% RSLogix 500 project Project_8.RSS, saved by version 8.30.00.16 %
PROJECT "UNTITLED"    % processor: Bul.1763 MicroLogix 1100 Series B %

PROGRAM FILES
  LAD 2 "MAIN"  4 rungs
  LAD 3 "IO"  3 rungs
  LAD 4 "CTL4%-15%"  7 rungs
  LAD 5 "CTL15%-30%"  7 rungs

DATA FILES
  O0 OUTPUT  4 elements
  I1 INPUT  6 elements
  S2 STATUS  66 elements
  B3 BINARY  3 elements
  T4 TIMER  4 elements
  C5 COUNTER  1 elements
  R6 CONTROL  1 elements
  N7 INTEGER  7 elements
  F8 FLOAT  1 elements

LADDER 2 "MAIN"
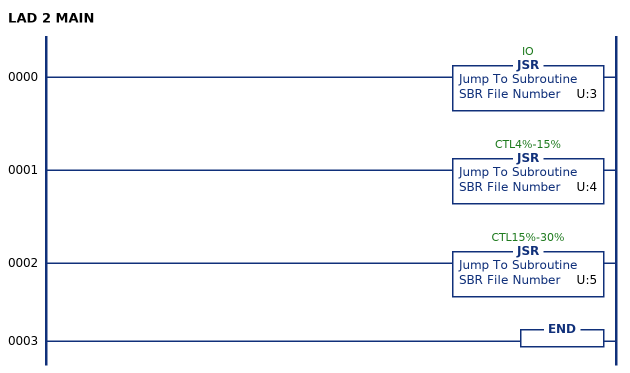
% Rung: 0 %
SOR JSR U:3 EOR
%   U:3  "IO" %
% Rung: 1 %
SOR JSR U:4 EOR
%   U:4  "CTL4%-15%" %
% Rung: 2 %
SOR JSR U:5 EOR
%   U:5  "CTL15%-30%" %
% Rung: 3 %
SOR END EOR

LADDER 3 "IO"
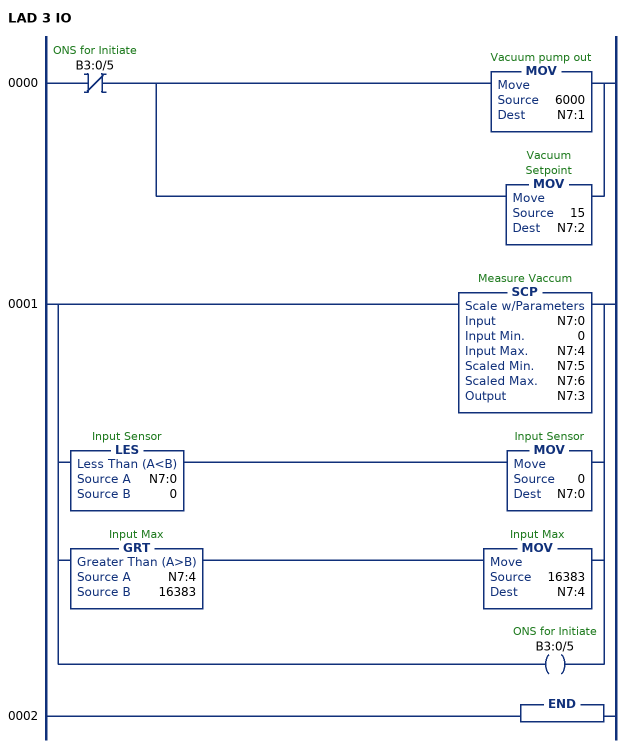
% Rung: 0 %
SOR XIO B3:0/5 BST MOV 6000 N7:1 NXB MOV 15 N7:2 BND EOR
%   B3:0/5  "ONS for Initiate" %
%   N7:1  "Vacuum pump out" %
%   N7:2  "Vacuum Setpoint" %
% Rung: 1 %
SOR BST SCP N7:0 0 N7:4 N7:5 N7:6 N7:3 NXB LES N7:0 0 MOV 0 N7:0 NXB GRT N7:4 16383 MOV 16383 N7:4 NXB OTE B3:0/5 BND EOR
%   N7:0  "Input Sensor" %
%   N7:4  "Input Max" %
%   N7:5  "Scale Min" %
%   N7:6  "Scale Max" %
%   N7:3  "Measure Vaccum" %
%   B3:0/5  "ONS for Initiate" %
% Rung: 2 %
SOR END EOR

LADDER 4 "CTL4%-15%"
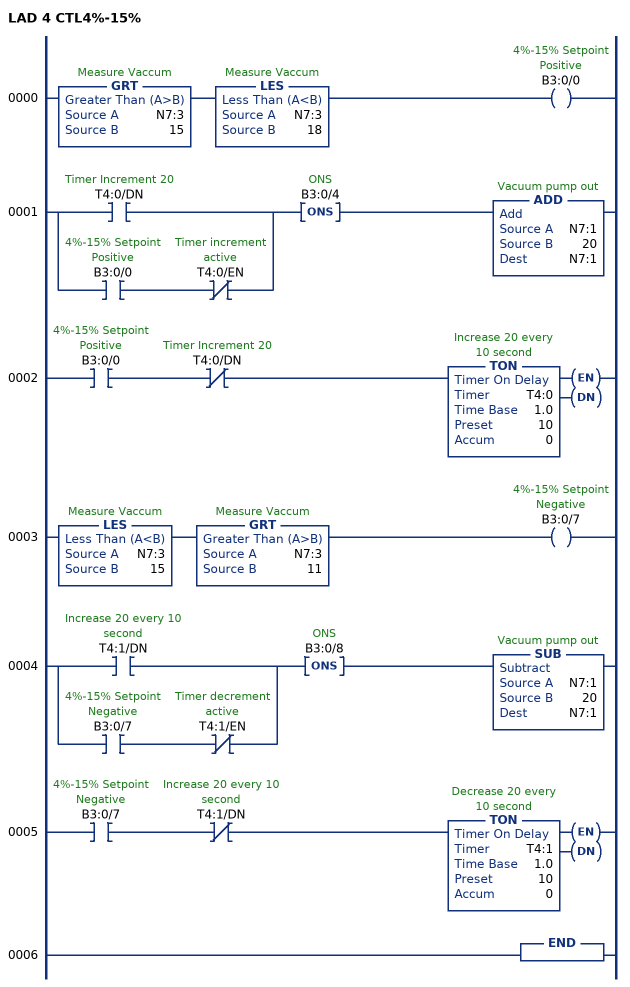
% Rung: 0 %
SOR GRT N7:3 15 LES N7:3 18 OTE B3:0/0 EOR
%   N7:3  "Measure Vaccum" %
%   B3:0/0  "4%-15% Setpoint Positive" %
% Rung: 1 %
SOR BST XIC T4:0/DN NXB XIC B3:0/0 XIO T4:0/EN BND ONS B3:0/4 ADD N7:1 20 N7:1 EOR
%   T4:0/DN  "Timer Increment 20" %
%   B3:0/0  "4%-15% Setpoint Positive" %
%   T4:0/EN  "Timer increment active" %
%   B3:0/4  "ONS" %
%   N7:1  "Vacuum pump out" %
% Rung: 2 %
SOR XIC B3:0/0 XIO T4:0/DN TON T4:0 1.0 10 0 EOR
%   B3:0/0  "4%-15% Setpoint Positive" %
%   T4:0/DN  "Timer Increment 20" %
%   T4:0  "Increase 20 every 10 second" %
% Rung: 3 %
SOR LES N7:3 15 GRT N7:3 11 OTE B3:0/7 EOR
%   N7:3  "Measure Vaccum" %
%   B3:0/7  "4%-15% Setpoint Negative" %
% Rung: 4 %
SOR BST XIC T4:1/DN NXB XIC B3:0/7 XIO T4:1/EN BND ONS B3:0/8 SUB N7:1 20 N7:1 EOR
%   T4:1/DN  "Increase 20 every 10 second" %
%   B3:0/7  "4%-15% Setpoint Negative" %
%   T4:1/EN  "Timer decrement active" %
%   B3:0/8  "ONS" %
%   N7:1  "Vacuum pump out" %
% Rung: 5 %
SOR XIC B3:0/7 XIO T4:1/DN TON T4:1 1.0 10 0 EOR
%   B3:0/7  "4%-15% Setpoint Negative" %
%   T4:1/DN  "Increase 20 every 10 second" %
%   T4:1  "Decrease 20 every 10 second" %
% Rung: 6 %
SOR END EOR

LADDER 5 "CTL15%-30%"
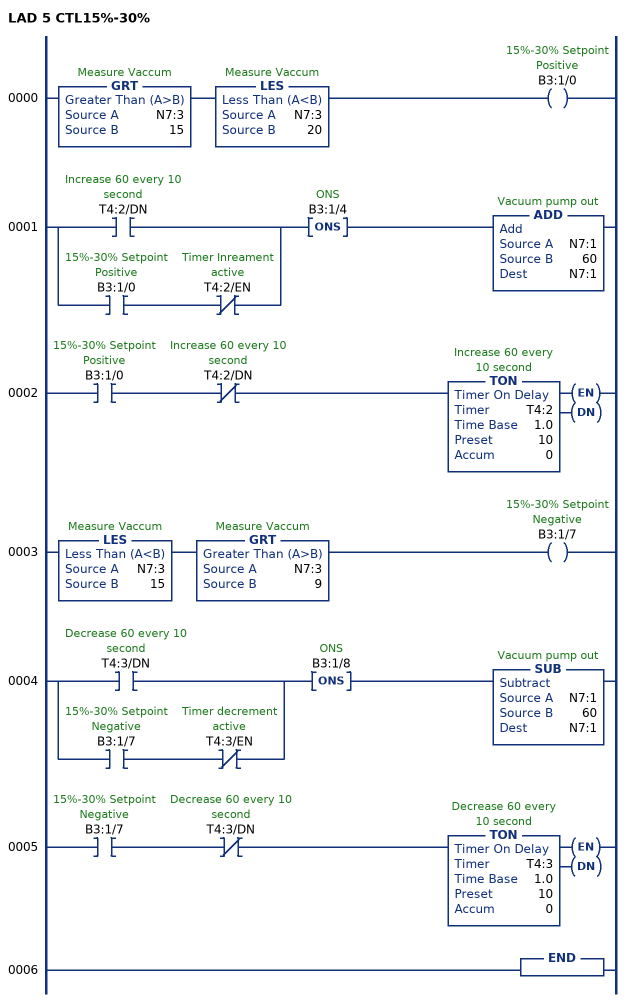
% Rung: 0 %
SOR GRT N7:3 15 LES N7:3 20 OTE B3:1/0 EOR
%   N7:3  "Measure Vaccum" %
%   B3:1/0  "15%-30% Setpoint Positive" %
% Rung: 1 %
SOR BST XIC T4:2/DN NXB XIC B3:1/0 XIO T4:2/EN BND ONS B3:1/4 ADD N7:1 60 N7:1 EOR
%   T4:2/DN  "Increase 60 every 10 second" %
%   B3:1/0  "15%-30% Setpoint Positive" %
%   T4:2/EN  "Timer Inreament active" %
%   B3:1/4  "ONS" %
%   N7:1  "Vacuum pump out" %
% Rung: 2 %
SOR XIC B3:1/0 XIO T4:2/DN TON T4:2 1.0 10 0 EOR
%   B3:1/0  "15%-30% Setpoint Positive" %
%   T4:2/DN  "Increase 60 every 10 second" %
%   T4:2  "Increase 60 every 10 second" %
% Rung: 3 %
SOR LES N7:3 15 GRT N7:3 9 OTE B3:1/7 EOR
%   N7:3  "Measure Vaccum" %
%   B3:1/7  "15%-30% Setpoint Negative" %
% Rung: 4 %
SOR BST XIC T4:3/DN NXB XIC B3:1/7 XIO T4:3/EN BND ONS B3:1/8 SUB N7:1 60 N7:1 EOR
%   T4:3  "Decrease 60 every 10 second" %
%   B3:1/7  "15%-30% Setpoint Negative" %
%   T4:3/EN  "Timer decrement active" %
%   B3:1/8  "ONS" %
%   N7:1  "Vacuum pump out" %
% Rung: 5 %
SOR XIC B3:1/7 XIO T4:3/DN TON T4:3 1.0 10 0 EOR
%   B3:1/7  "15%-30% Setpoint Negative" %
%   T4:3  "Decrease 60 every 10 second" %
% Rung: 6 %
SOR END EOR

OTHER DOCUMENTED ADDRESSES
  B3:0/1  "ONS"
  B3:0/2  "Timer"
  B3:0/3  "test"
  B3:0/6  "Reset Timer"

DATA TABLE (non-zero values as saved)
DATA T4
% .PRE .ACC %
% T4:0 % 10 0
% T4:1 % 10 0
% T4:2 % 10 0
% T4:3 % 10 0
DATA N7
% N7:0 % 10000 0 0 0 16383 0 30
